FUNCTION_BLOCK FB_Axis_Discrete_HomeToExternalForce EXTENDS FB_Axis_HomeToExternalForceFeedback
VAR_INPUT
END_VAR
VAR_OUTPUT
END_VAR
VAR
	//If preferred, initialize upper limit to a value less than the lower limit to prevent operation until proper soft limits have been configured
	fLowerTravelLimit			: LREAL := -1.7976931348623158E+308; //(Minimum LREAL value)
	fUpperTravelLimit			: LREAL := 1.7976931348623158E+308;	//(Maximum LREAL value)
	fPosition_1					: LREAL;
	fPosition_2					: LREAL;
	fPosition_3					: LREAL;
	
END_VAR

PROPERTY LowerTravelLimit : LREAL
GET
LowerTravelLimit := fLowerTravelLimit;
END_GET
SET
fLowerTravelLimit := LowerTravelLimit;
END_SET
END_PROPERTY

METHOD Monitoring : BOOL
VAR_INPUT
END_VAR
//Monitor soft travel limits
IF fPosition >= fUpperTravelLimit AND fPositionSetpoint > fUpperTravelLimit THEN
	Inhibit();
	//TODO: log specific message for soft limit reached
END_IF

IF fPosition <= fLowerTravelLimit AND fPositionSetpoint < fLowerTravelLimit THEN
	Inhibit();
	//TODO: log specific message for soft limit reached
END_IF

IF  fOverride = 0 AND fPositionSetpoint < fUpperTravelLimit AND fPositionSetpoint > fLowerTravelLimit THEN
	Uninhibit();
	//TODO: log specific message for soft limit reached
END_IF

SUPER^.Monitoring();		//Called last to allow the bReady bit to be evaluated after all error checking is done
END_METHOD

PROPERTY TargetPosition_1 : LREAL
GET
TargetPosition_1 := fPosition_1;
END_GET
SET
fPosition_1 := TargetPosition_1;
END_SET
END_PROPERTY

PROPERTY TargetPosition_2 : LREAL
GET
TargetPosition_2 := fPosition_2;
END_GET
SET
fPosition_2 := TargetPosition_2;
END_SET
END_PROPERTY

PROPERTY TargetPosition_3 : LREAL
GET
TargetPosition_3 := fPosition_3;
END_GET
SET
fPosition_3 := TargetPosition_3;
END_SET
END_PROPERTY

PROPERTY UpperTravelLimit : LREAL
GET
UpperTravelLimit := fUpperTravelLimit;
END_GET
SET
fUpperTravelLimit := UpperTravelLimit;
END_SET
END_PROPERTY

END_FUNCTION_BLOCK

(* stored: Version 1.1.0.1, ProductVersion 3.1.4024.9
   POU FB_Axis_Discrete_HomeToExternalForce: Id {2424e970-a6a9-41ec-8de7-dfd65a5be1e6}, SpecialFunc None
   Folder 01_SUPER_Overrides: Id {8bd99d59-60b9-419d-8640-6eb28ef92ffd}
   Folder 02_ITF_Axis_Discrete: Id {81a2e083-ae97-489c-adf0-0e60e4967c2c}
   Property LowerTravelLimit: Id {4a129ee9-0d1d-4140-bca5-cd14adc01819}
   Get Get: Id {ec5d9a54-ce47-451e-957a-a0e8fe75e047}
   Set Set: Id {cdd2a299-f5a2-489a-aefa-7c2a25cb3356}
   Method Monitoring: Id {48a54ca3-391a-480a-a2de-5038a1059daa}
   Property TargetPosition_1: Id {a972d644-c7dd-43f3-9398-b67ece98d19c}
   Get Get: Id {64d8a513-a91e-45a8-a836-740617cbc3f8}
   Set Set: Id {e09d3743-74fe-41dd-b702-b822650f5bc4}
   Property TargetPosition_2: Id {b23e4a70-d4ad-4067-b7ba-95261838e3af}
   Get Get: Id {9970c4da-fd15-44de-b4e2-1be335312192}
   Set Set: Id {48d2f6fe-972e-44a5-a7bb-06808c72e604}
   Property TargetPosition_3: Id {20e3cf89-d928-4cca-b21e-3ac246aa968e}
   Get Get: Id {aa1fad92-ab28-4d46-b759-448fe339c3d2}
   Set Set: Id {36bc4dbc-ed47-4e4d-8416-7eb214c6408b}
   Property UpperTravelLimit: Id {6a86d957-5414-4aa2-b4c9-274e2e6810ab}
   Get Get: Id {b56f1dbb-75ee-439c-8849-11f2702afaff}
   Set Set: Id {237fa5a5-8049-44a0-a82d-5a94fe6eb0d4} *)
